FUNCTION_BLOCK FB_mb_to_val
VAR_INPUT
	xi: REAL:=0;
	i_hi: REAL:=20.0;
	cal_dc_offset: REAL :=0;
	y_h: REAL:= 0.0;
END_VAR

VAR_OUTPUT
	y: REAL;
END_VAR

VAR
	xi_cal: REAL;
END_VAR



xi_cal := xi - cal_dc_offset;
y:=y_h*xi_cal/i_hi;
IF y>y_h THEN
	y:=y_h;
ELSIF y < 0 THEN
	y:=0.0;	
END_IF

END_FUNCTION_BLOCK

(* stored: Version 1.1.0.1, ProductVersion 3.1.0.36
   POU FB_mb_to_val: Id {bf0f1eb1-fac2-48c0-84b3-2ba62933f004}, SpecialFunc None *)
